FUNCTION RDM : REAL
VAR_INPUT
	last : REAL;
END_VAR
VAR
	tn : DWORD;
	tc : INT;
END_VAR


(*
version 1.9	10. mar. 2009
programmer 	hugo
tested by		tobias

this function calculates a pseudo random number
to generate the number it reads the sps timer and calculates a random number between 0 and 1:
in order to use rdm more then once within one sps cycle it need to be called with different seed numbers LAST.

*)

tn := T_PLC_MS();
tc := BIT_COUNT(tn);
tn.31 := tn.2;
tn.30 := tn.5;
tn.29 := tn.4;
tn.28 := tn.1;
tn.27 := tn.0;
tn.26 := tn.7;
tn.25 := tn.6;
tn.24 := tn.3;
tn := ROL(tn,BIT_COUNT(tn)) OR 16#80000001;
tn := tn MOD 71474513 + INT_TO_DWORD(tc + 77);
RDM := FRACT(DWORD_TO_REAL(tn) / 10000000.0 * (math.E - LIMIT(0.0,last,1.0)));


(*
pt := ADR(temp);
pt^ := (T_PLC_MS() AND 16#007FFFFF) OR 16#3D000000;
RDM := fract(modR(temp*e+pi1, PI1-last) + modR(temp*PI1+e + last,e-last));
*)

(* revision history
hm		16. jan 2007		rev 1.0
	original version

hm		11. nov 2007		rev 1.1
	changed time() into t_plc_ms()

hm		20. nov 2007		rev 1.2
	changed code of temp calculation to avoid overflow in modr due to resuclt would not fit DINT for high timeer values

hm		5. jan 2008		rev 1.3
	changed calculation of temp to avoid problem with high values of t_plc_ms

hm		2. feb 2008		rev 1.4
	changed algorithm to avoind non iec functions and guarantee more randomness

hm	10. mar. 2008		rev 1.5
	make sure last will be between 0 and 1 to avoid invalid results

hm	16. mar. 2008		rev 1.6
	added conversion for tc to avoid warnings under codesys 3.0

hm	18. may. 2008		rev 1.7
	changed constant E to E1

hm	18. oct. 2008		rev 1.8
	using math constants

hm	10. mar. 2009		rev 1.9
	real constants updated to new systax using dot

*)

END_FUNCTION

(* stored: Version 1.1.0.1, ProductVersion 3.1.4022.7
   POU RDM: Id {db8f0d5e-0d82-45fc-99e9-94665647aed9}, SpecialFunc None *)
